(* Schneider Machine Expert - Basic project Push Button Program with switching, file version 2.9.0.0 *)
(* ProjectInformations: Name=New project *)

HARDWARE
  Cpu 0: TM221C24R
  EthernetConfiguration: NetworkName=M221, IpAllocationMode=FixedAddress, IpAddress=0.0.0.0, SubnetMask=0.0.0.0
  SerialLineConfiguration: Baud=Baud19200, Parity=ParityEven, DataBits=DataBits8, StopBits=StopBits1, PhysicalMedium=PhysicalMediumRs485, SlaveId=1, Addressing=SlaveAddressing
  MastTask: UsePeriodScanMode=false, PeriodScan=100
  FastTask: Period=255
  CpuBehavior: StartingMode=StartAsPreviousState, AutoSaveRamOnEeprom=true, WatchdogPeriod=250

SYMBOLS  (address, symbol, comment, settings)
  %M0       MEMORY_BIT_1
  %M1       MEMORY_BIT_2
  %I0.0     SWITCH_1
  %Q0.0     OUTPUT

POU New POU
  (* SectionNumber=1 *)

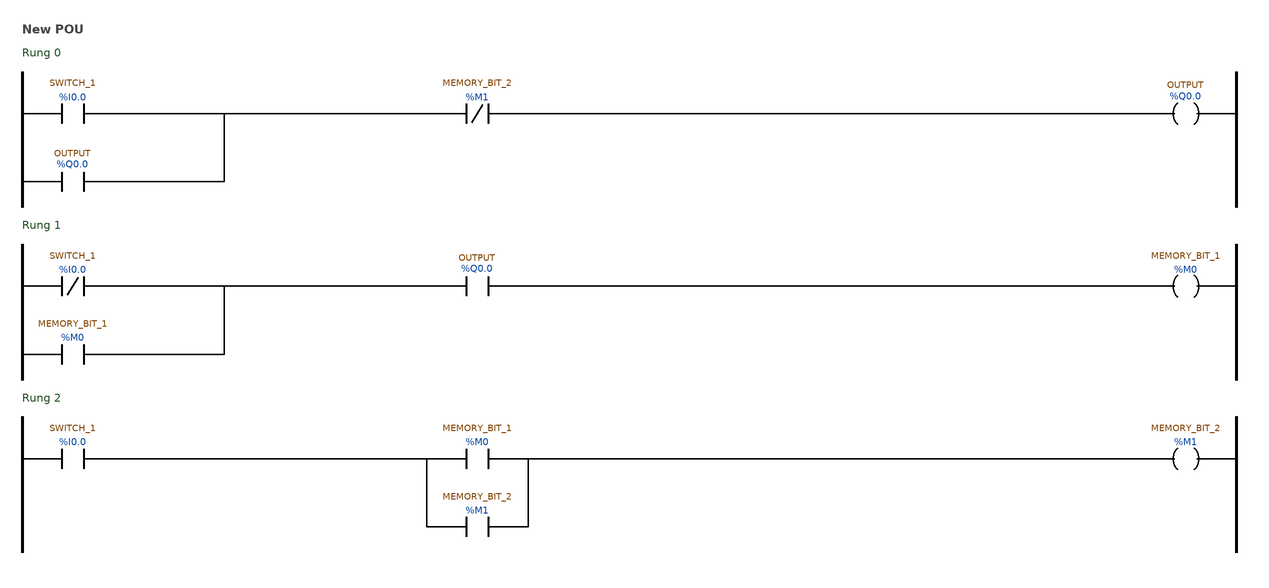

// Rung 0
  LD %I0.0                (* SWITCH_1 *)
  OR %Q0.0                (* OUTPUT *)
  ANDN %M1                (* MEMORY_BIT_2 *)
  ST %Q0.0                (* OUTPUT *)
  // as ST:
  //   OUTPUT := (SWITCH_1 OR OUTPUT) AND NOT MEMORY_BIT_2;

// Rung 1
  LDN %I0.0               (* SWITCH_1 *)
  OR %M0                  (* MEMORY_BIT_1 *)
  AND %Q0.0               (* OUTPUT *)
  ST %M0                  (* MEMORY_BIT_1 *)
  // as ST:
  //   MEMORY_BIT_1 := (NOT SWITCH_1 OR MEMORY_BIT_1) AND OUTPUT;

// Rung 2
  LD %I0.0                (* SWITCH_1 *)
  AND( %M0                (* MEMORY_BIT_1 *)
  OR %M1                  (* MEMORY_BIT_2 *)
  )
  ST %M1                  (* MEMORY_BIT_2 *)
  // as ST:
  //   MEMORY_BIT_2 := SWITCH_1 AND (MEMORY_BIT_1 OR MEMORY_BIT_2);
